(* CoDeSys 2.3 export: GVL_ADSCLIENTTESTS.EXP *)

(* Global variable list: AdsClientTests/GVL_AdsClientTests *)
VAR_GLOBAL
	VERSION	: STRING := '2.0.0';
	IsReset 		: BOOL := TRUE;
	IsTestProject 	: BOOL := TRUE;
	IsRunning 	: BOOL;
	TestPointer 	: POINTER TO BOOL; (*//FOR 32/64bit check*)
	IsTc2 		: BOOL := TRUE;
END_VAR
